// TIA Portal V16 export
// export: Created 2021-06-01T00:01:15.1519553Z, ExportSetting WithDefaults, DisplayName Totally Integrated Automation Portal, DisplayVersion V16 Update 4, DisplayName TIA Portal Version Control Interface, DisplayVersion V16 Update 2, DisplayName TIA Portal Openness, DisplayVersion V16 Update 4, DisplayName STEP 7 Professional, DisplayVersion V16 Update 4, DisplayName STEP 7 Safety, DisplayVersion V16, DisplayName WinCC Advanced, DisplayVersion V16 Update 4
FUNCTION_BLOCK "Block_1"   // FB2, F_FBD
{ S7_Optimized_Access := 'TRUE' }
VERSION : 0.1
// stored: AutoNumber true, IsIECCheckEnabled false, UDAEnableTagReadback false
   VAR_INPUT
      "a" : Bool;
   END_VAR
   VAR_OUTPUT
      out0 : Bool;
      out1 : Bool;
   END_VAR
   VAR_TEMP
      t0 : Bool;
      ton : Bool;
   END_VAR
   VAR CONSTANT
      ALWAYS_FALSE : Bool := false;
   END_VAR
BEGIN

REGION Network 1
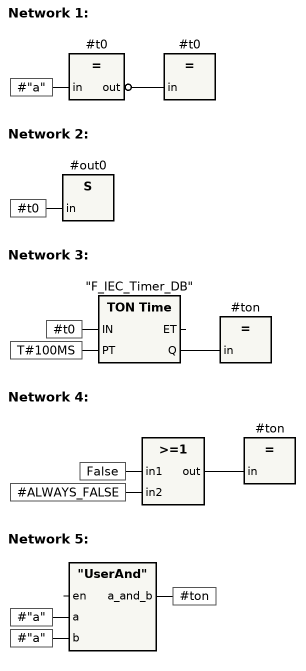
   #t0 := #"a";
   #t0 := NOT #"a";
END_REGION

REGION Network 2
   IF #t0 THEN #out0 := TRUE; END_IF;
END_REGION

REGION Network 3
   "F_IEC_Timer_DB".TON(IN := #t0, PT := T#100MS);
   #ton := "F_IEC_Timer_DB".Q;
END_REGION

REGION Network 4
   #ton := False OR #ALWAYS_FALSE;
END_REGION

REGION Network 5
   "UserAnd"("a" := #"a", "b" := #"a", a_and_b => #ton);
END_REGION
END_FUNCTION_BLOCK
